% RSLogix 500 project IIS REV 1.0. 4.29.16.RSS, saved by version 10.00.00.00 %
PROJECT "IISM1200"    % processor: MicroLogix 1200 %

PROGRAM FILES
  LAD 2 "MAIN_PROG"  27 rungs

DATA FILES
  O0 OUTPUT  4 elements
  I1 INPUT  4 elements
  S2 STATUS  66 elements
  B3 BINARY  2 elements
  T4 TIMER  4 elements
  C5 COUNTER  1 elements
  R6 CONTROL  1 elements
  N7 INTEGER  1 elements
  F8 FLOAT  1 elements

LADDER 2 "MAIN_PROG"
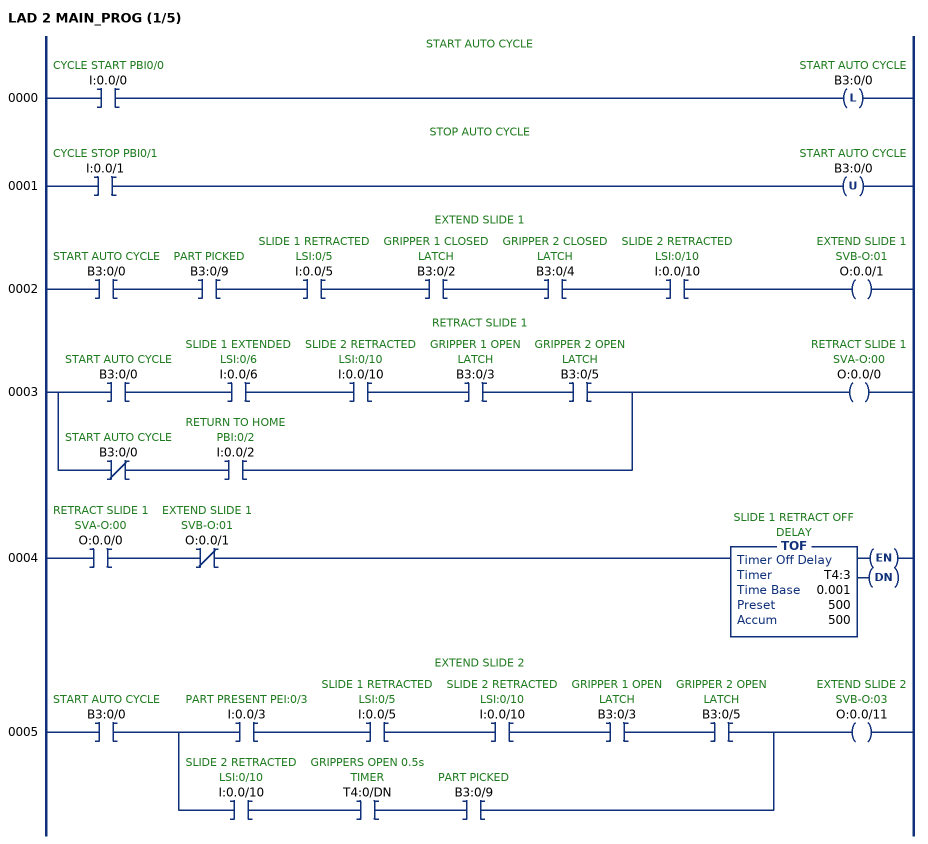
% Rung: 0 %
% START AUTO CYCLE %
SOR XIC I:0.0/0 OTL B3:0/0 EOR
%   I:0.0/0  "CYCLE START PBI0/0" %
%   B3:0/0  "START AUTO CYCLE" %
% Rung: 1 %
% STOP AUTO CYCLE %
SOR XIC I:0.0/1 OTU B3:0/0 EOR
%   I:0.0/1  "CYCLE STOP PBI0/1" %
%   B3:0/0  "START AUTO CYCLE" %
% Rung: 2 %
% EXTEND SLIDE 1 %
SOR XIC B3:0/0 XIC B3:0/9 XIC I:0.0/5 XIC B3:0/2 XIC B3:0/4 XIC I:0.0/10 OTE O:0.0/1 EOR
%   B3:0/0  "START AUTO CYCLE" %
%   B3:0/9  "PART PICKED" %
%   I:0.0/5  "SLIDE 1 RETRACTED LSI:0/5" %
%   B3:0/2  "GRIPPER 1 CLOSED LATCH" %
%   B3:0/4  "GRIPPER 2 CLOSED LATCH" %
%   I:0.0/10  "SLIDE 2 RETRACTED LSI:0/10" %
%   O:0.0/1  "EXTEND SLIDE 1 SVB-O:01" %
% Rung: 3 %
% RETRACT SLIDE 1 %
SOR BST XIC B3:0/0 XIC I:0.0/6 XIC I:0.0/10 XIC B3:0/3 XIC B3:0/5 NXB XIO B3:0/0 XIC I:0.0/2 BND OTE O:0.0/0 EOR
%   B3:0/0  "START AUTO CYCLE" %
%   I:0.0/6  "SLIDE 1 EXTENDED LSI:0/6" %
%   I:0.0/10  "SLIDE 2 RETRACTED LSI:0/10" %
%   B3:0/3  "GRIPPER 1 OPEN LATCH" %
%   B3:0/5  "GRIPPER 2 OPEN LATCH" %
%   I:0.0/2  "RETURN TO HOME PBI:0/2" %
%   O:0.0/0  "RETRACT SLIDE 1 SVA-O:00" %
% Rung: 4 %
SOR XIC O:0.0/0 XIO O:0.0/1 TOF T4:3 0.001 500 500 EOR
%   O:0.0/0  "RETRACT SLIDE 1 SVA-O:00" %
%   O:0.0/1  "EXTEND SLIDE 1 SVB-O:01" %
%   T4:3  "SLIDE 1 RETRACT OFF DELAY" %
% Rung: 5 %
% EXTEND SLIDE 2 %
SOR XIC B3:0/0 BST XIC I:0.0/3 XIC I:0.0/5 XIC I:0.0/10 XIC B3:0/3 XIC B3:0/5 NXB XIC I:0.0/10 XIC T4:0/DN XIC B3:0/9 BND OTE O:0.0/11 EOR
%   B3:0/0  "START AUTO CYCLE" %
%   I:0.0/3  "PART PRESENT PEI:0/3" %
%   I:0.0/5  "SLIDE 1 RETRACTED LSI:0/5" %
%   I:0.0/10  "SLIDE 2 RETRACTED LSI:0/10" %
%   B3:0/3  "GRIPPER 1 OPEN LATCH" %
%   B3:0/5  "GRIPPER 2 OPEN LATCH" %
%   T4:0  "GRIPPERS OPEN 0.5s TIMER" %
%   B3:0/9  "PART PICKED" %
%   O:0.0/11  "EXTEND SLIDE 2 SVB-O:03" %

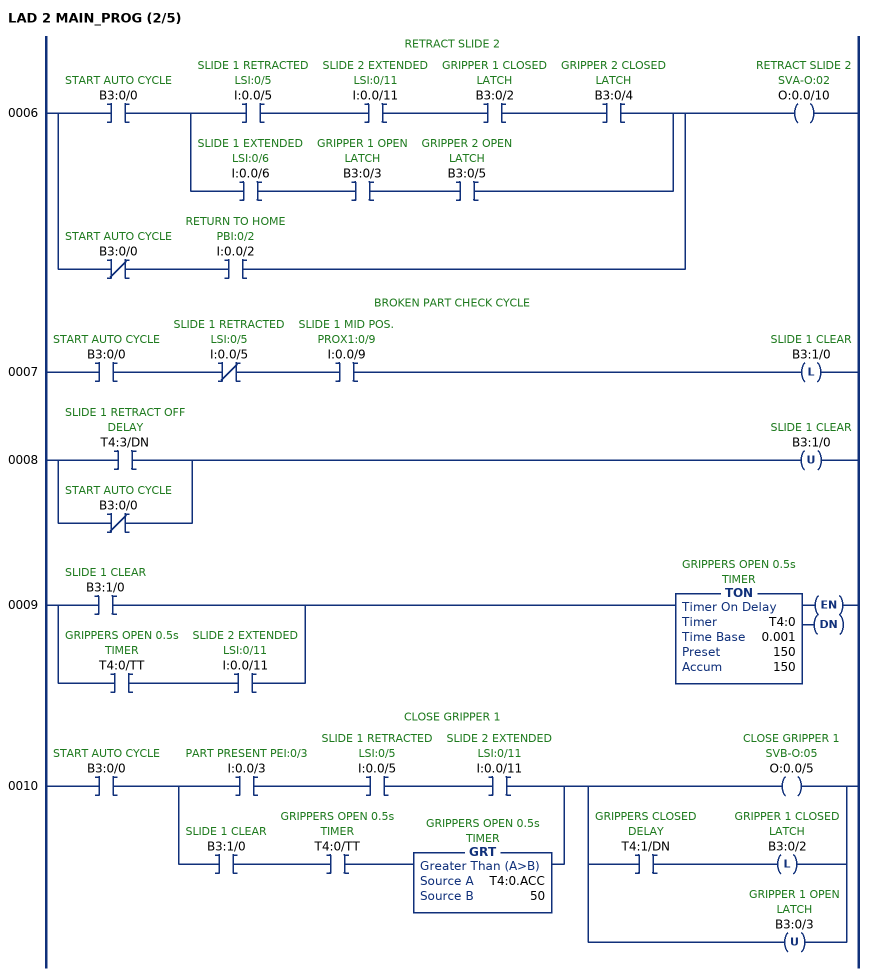
% Rung: 6 %
% RETRACT SLIDE 2 %
SOR BST XIC B3:0/0 BST XIC I:0.0/5 XIC I:0.0/11 XIC B3:0/2 XIC B3:0/4 NXB XIC I:0.0/6 XIC B3:0/3 XIC B3:0/5 BND NXB XIO B3:0/0 XIC I:0.0/2 BND OTE O:0.0/10 EOR
%   B3:0/0  "START AUTO CYCLE" %
%   I:0.0/5  "SLIDE 1 RETRACTED LSI:0/5" %
%   I:0.0/11  "SLIDE 2 EXTENDED LSI:0/11" %
%   B3:0/2  "GRIPPER 1 CLOSED LATCH" %
%   B3:0/4  "GRIPPER 2 CLOSED LATCH" %
%   I:0.0/6  "SLIDE 1 EXTENDED LSI:0/6" %
%   B3:0/3  "GRIPPER 1 OPEN LATCH" %
%   B3:0/5  "GRIPPER 2 OPEN LATCH" %
%   I:0.0/2  "RETURN TO HOME PBI:0/2" %
%   O:0.0/10  "RETRACT SLIDE 2 SVA-O:02" %
% Rung: 7 %
% BROKEN PART CHECK CYCLE %
SOR XIC B3:0/0 XIO I:0.0/5 XIC I:0.0/9 OTL B3:1/0 EOR
%   B3:0/0  "START AUTO CYCLE" %
%   I:0.0/5  "SLIDE 1 RETRACTED LSI:0/5" %
%   I:0.0/9  "SLIDE 1 MID POS. PROX1:0/9" %
%   B3:1/0  "SLIDE 1 CLEAR" %
% Rung: 8 %
SOR BST XIC T4:3/DN NXB XIO B3:0/0 BND OTU B3:1/0 EOR
%   T4:3  "SLIDE 1 RETRACT OFF DELAY" %
%   B3:0/0  "START AUTO CYCLE" %
%   B3:1/0  "SLIDE 1 CLEAR" %
% Rung: 9 %
SOR BST XIC B3:1/0 NXB XIC T4:0/TT XIC I:0.0/11 BND TON T4:0 0.001 150 150 EOR
%   B3:1/0  "SLIDE 1 CLEAR" %
%   T4:0  "GRIPPERS OPEN 0.5s TIMER" %
%   I:0.0/11  "SLIDE 2 EXTENDED LSI:0/11" %
% Rung: 10 %
% CLOSE GRIPPER 1 %
SOR XIC B3:0/0 BST XIC I:0.0/3 XIC I:0.0/5 XIC I:0.0/11 NXB XIC B3:1/0 XIC T4:0/TT GRT T4:0.ACC 50 BND BST OTE O:0.0/5 NXB XIC T4:1/DN OTL B3:0/2 NXB OTU B3:0/3 BND EOR
%   B3:0/0  "START AUTO CYCLE" %
%   I:0.0/3  "PART PRESENT PEI:0/3" %
%   I:0.0/5  "SLIDE 1 RETRACTED LSI:0/5" %
%   I:0.0/11  "SLIDE 2 EXTENDED LSI:0/11" %
%   B3:1/0  "SLIDE 1 CLEAR" %
%   T4:0  "GRIPPERS OPEN 0.5s TIMER" %
%   O:0.0/5  "CLOSE GRIPPER 1 SVB-O:05" %
%   T4:1/DN  "GRIPPERS CLOSED DELAY" %
%   B3:0/2  "GRIPPER 1 CLOSED LATCH" %
%   B3:0/3  "GRIPPER 1 OPEN LATCH" %

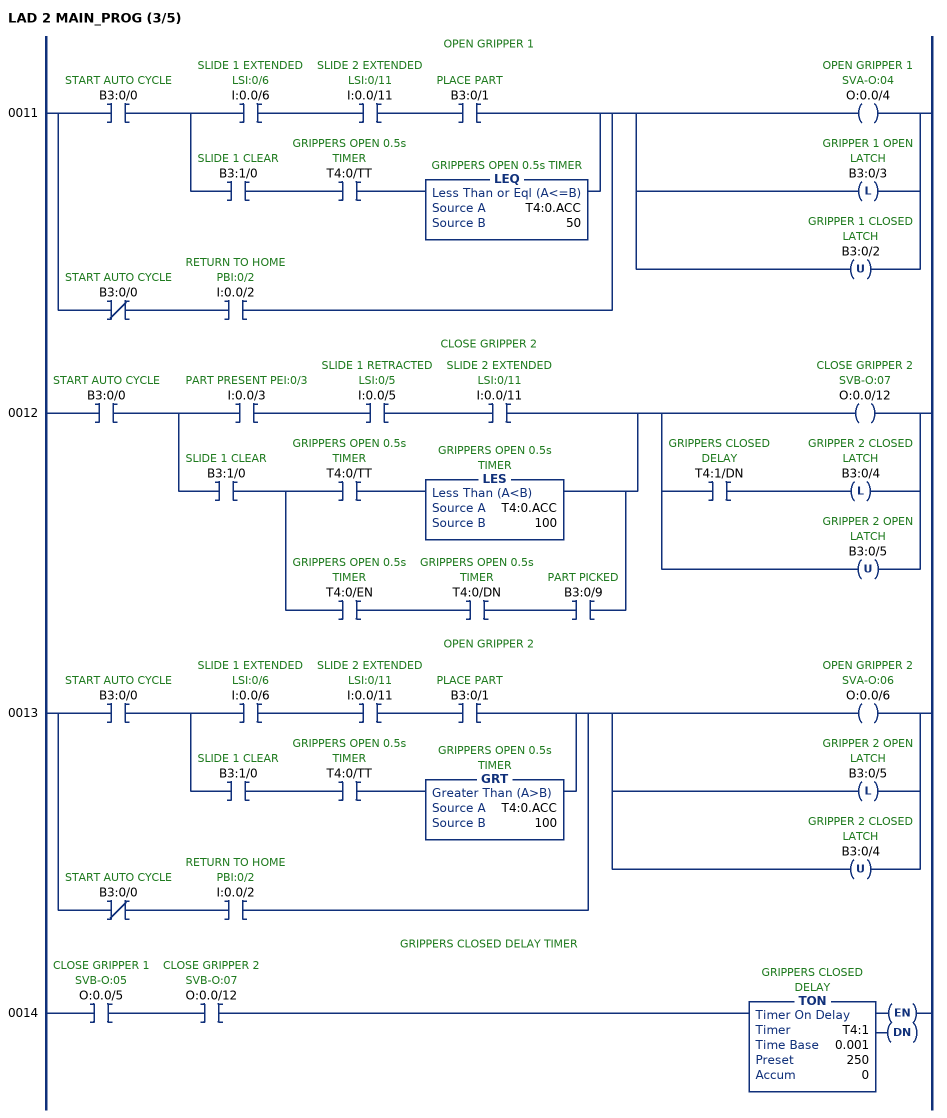
% Rung: 11 %
% OPEN GRIPPER 1 %
SOR BST XIC B3:0/0 BST XIC I:0.0/6 XIC I:0.0/11 XIC B3:0/1 NXB XIC B3:1/0 XIC T4:0/TT LEQ T4:0.ACC 50 BND NXB XIO B3:0/0 XIC I:0.0/2 BND BST OTE O:0.0/4 NXB OTL B3:0/3 NXB OTU B3:0/2 BND EOR
%   B3:0/0  "START AUTO CYCLE" %
%   I:0.0/6  "SLIDE 1 EXTENDED LSI:0/6" %
%   I:0.0/11  "SLIDE 2 EXTENDED LSI:0/11" %
%   B3:0/1  "PLACE PART" %
%   B3:1/0  "SLIDE 1 CLEAR" %
%   T4:0  "GRIPPERS OPEN 0.5s TIMER" %
%   I:0.0/2  "RETURN TO HOME PBI:0/2" %
%   O:0.0/4  "OPEN GRIPPER 1 SVA-O:04" %
%   B3:0/3  "GRIPPER 1 OPEN LATCH" %
%   B3:0/2  "GRIPPER 1 CLOSED LATCH" %
% Rung: 12 %
% CLOSE GRIPPER 2 %
SOR XIC B3:0/0 BST XIC I:0.0/3 XIC I:0.0/5 XIC I:0.0/11 NXB XIC B3:1/0 BST XIC T4:0/TT LES T4:0.ACC 100 NXB XIC T4:0/EN XIC T4:0/DN XIC B3:0/9 BND BND BST OTE O:0.0/12 NXB XIC T4:1/DN OTL B3:0/4 NXB OTU B3:0/5 BND EOR
%   B3:0/0  "START AUTO CYCLE" %
%   I:0.0/3  "PART PRESENT PEI:0/3" %
%   I:0.0/5  "SLIDE 1 RETRACTED LSI:0/5" %
%   I:0.0/11  "SLIDE 2 EXTENDED LSI:0/11" %
%   B3:1/0  "SLIDE 1 CLEAR" %
%   T4:0  "GRIPPERS OPEN 0.5s TIMER" %
%   B3:0/9  "PART PICKED" %
%   O:0.0/12  "CLOSE GRIPPER 2 SVB-O:07" %
%   T4:1/DN  "GRIPPERS CLOSED DELAY" %
%   B3:0/4  "GRIPPER 2 CLOSED LATCH" %
%   B3:0/5  "GRIPPER 2 OPEN LATCH" %
% Rung: 13 %
% OPEN GRIPPER 2 %
SOR BST XIC B3:0/0 BST XIC I:0.0/6 XIC I:0.0/11 XIC B3:0/1 NXB XIC B3:1/0 XIC T4:0/TT GRT T4:0.ACC 100 BND NXB XIO B3:0/0 XIC I:0.0/2 BND BST OTE O:0.0/6 NXB OTL B3:0/5 NXB OTU B3:0/4 BND EOR
%   B3:0/0  "START AUTO CYCLE" %
%   I:0.0/6  "SLIDE 1 EXTENDED LSI:0/6" %
%   I:0.0/11  "SLIDE 2 EXTENDED LSI:0/11" %
%   B3:0/1  "PLACE PART" %
%   B3:1/0  "SLIDE 1 CLEAR" %
%   T4:0  "GRIPPERS OPEN 0.5s TIMER" %
%   I:0.0/2  "RETURN TO HOME PBI:0/2" %
%   O:0.0/6  "OPEN GRIPPER 2 SVA-O:06" %
%   B3:0/5  "GRIPPER 2 OPEN LATCH" %
%   B3:0/4  "GRIPPER 2 CLOSED LATCH" %
% Rung: 14 %
% GRIPPERS CLOSED DELAY TIMER %
SOR XIC O:0.0/5 XIC O:0.0/12 TON T4:1 0.001 250 0 EOR
%   O:0.0/5  "CLOSE GRIPPER 1 SVB-O:05" %
%   O:0.0/12  "CLOSE GRIPPER 2 SVB-O:07" %
%   T4:1  "GRIPPERS CLOSED DELAY" %

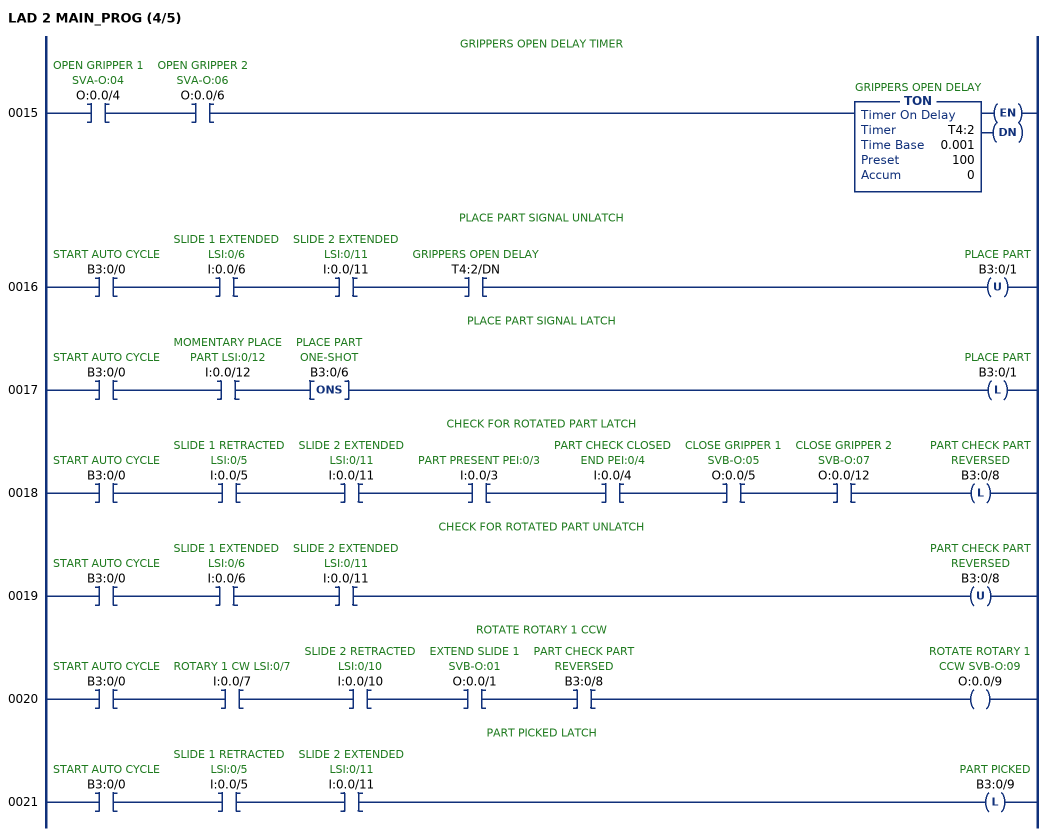
% Rung: 15 %
% GRIPPERS OPEN DELAY TIMER %
SOR XIC O:0.0/4 XIC O:0.0/6 TON T4:2 0.001 100 0 EOR
%   O:0.0/4  "OPEN GRIPPER 1 SVA-O:04" %
%   O:0.0/6  "OPEN GRIPPER 2 SVA-O:06" %
%   T4:2  "GRIPPERS OPEN DELAY" %
% Rung: 16 %
% PLACE PART SIGNAL UNLATCH %
SOR XIC B3:0/0 XIC I:0.0/6 XIC I:0.0/11 XIC T4:2/DN OTU B3:0/1 EOR
%   B3:0/0  "START AUTO CYCLE" %
%   I:0.0/6  "SLIDE 1 EXTENDED LSI:0/6" %
%   I:0.0/11  "SLIDE 2 EXTENDED LSI:0/11" %
%   T4:2  "GRIPPERS OPEN DELAY" %
%   B3:0/1  "PLACE PART" %
% Rung: 17 %
% PLACE PART SIGNAL LATCH %
SOR XIC B3:0/0 XIC I:0.0/12 ONS B3:0/6 OTL B3:0/1 EOR
%   B3:0/0  "START AUTO CYCLE" %
%   I:0.0/12  "MOMENTARY PLACE PART LSI:0/12" %
%   B3:0/6  "PLACE PART ONE-SHOT" %
%   B3:0/1  "PLACE PART" %
% Rung: 18 %
% CHECK FOR ROTATED PART LATCH %
SOR XIC B3:0/0 XIC I:0.0/5 XIC I:0.0/11 XIC I:0.0/3 XIC I:0.0/4 XIC O:0.0/5 XIC O:0.0/12 OTL B3:0/8 EOR
%   B3:0/0  "START AUTO CYCLE" %
%   I:0.0/5  "SLIDE 1 RETRACTED LSI:0/5" %
%   I:0.0/11  "SLIDE 2 EXTENDED LSI:0/11" %
%   I:0.0/3  "PART PRESENT PEI:0/3" %
%   I:0.0/4  "PART CHECK CLOSED END PEI:0/4" %
%   O:0.0/5  "CLOSE GRIPPER 1 SVB-O:05" %
%   O:0.0/12  "CLOSE GRIPPER 2 SVB-O:07" %
%   B3:0/8  "PART CHECK PART REVERSED" %
% Rung: 19 %
% CHECK FOR ROTATED PART UNLATCH %
SOR XIC B3:0/0 XIC I:0.0/6 XIC I:0.0/11 OTU B3:0/8 EOR
%   B3:0/0  "START AUTO CYCLE" %
%   I:0.0/6  "SLIDE 1 EXTENDED LSI:0/6" %
%   I:0.0/11  "SLIDE 2 EXTENDED LSI:0/11" %
%   B3:0/8  "PART CHECK PART REVERSED" %
% Rung: 20 %
% ROTATE ROTARY 1 CCW %
SOR XIC B3:0/0 XIC I:0.0/7 XIC I:0.0/10 XIC O:0.0/1 XIC B3:0/8 OTE O:0.0/9 EOR
%   B3:0/0  "START AUTO CYCLE" %
%   I:0.0/7  "ROTARY 1 CW LSI:0/7" %
%   I:0.0/10  "SLIDE 2 RETRACTED LSI:0/10" %
%   O:0.0/1  "EXTEND SLIDE 1 SVB-O:01" %
%   B3:0/8  "PART CHECK PART REVERSED" %
%   O:0.0/9  "ROTATE ROTARY 1 CCW SVB-O:09" %
% Rung: 21 %
% PART PICKED LATCH %
SOR XIC B3:0/0 XIC I:0.0/5 XIC I:0.0/11 OTL B3:0/9 EOR
%   B3:0/0  "START AUTO CYCLE" %
%   I:0.0/5  "SLIDE 1 RETRACTED LSI:0/5" %
%   I:0.0/11  "SLIDE 2 EXTENDED LSI:0/11" %
%   B3:0/9  "PART PICKED" %

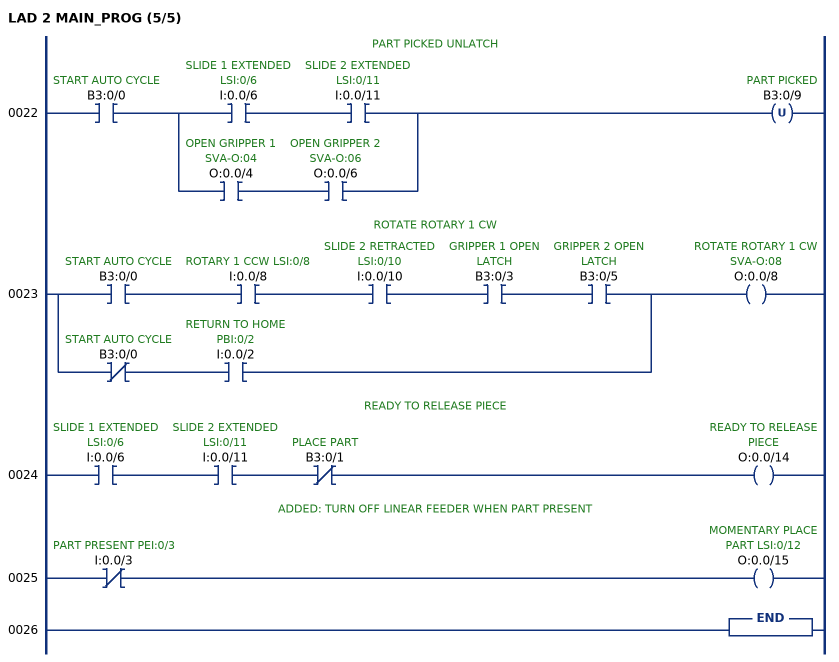
% Rung: 22 %
% PART PICKED UNLATCH %
SOR XIC B3:0/0 BST XIC I:0.0/6 XIC I:0.0/11 NXB XIC O:0.0/4 XIC O:0.0/6 BND OTU B3:0/9 EOR
%   B3:0/0  "START AUTO CYCLE" %
%   I:0.0/6  "SLIDE 1 EXTENDED LSI:0/6" %
%   I:0.0/11  "SLIDE 2 EXTENDED LSI:0/11" %
%   O:0.0/4  "OPEN GRIPPER 1 SVA-O:04" %
%   O:0.0/6  "OPEN GRIPPER 2 SVA-O:06" %
%   B3:0/9  "PART PICKED" %
% Rung: 23 %
% ROTATE ROTARY 1 CW %
SOR BST XIC B3:0/0 XIC I:0.0/8 XIC I:0.0/10 XIC B3:0/3 XIC B3:0/5 NXB XIO B3:0/0 XIC I:0.0/2 BND OTE O:0.0/8 EOR
%   B3:0/0  "START AUTO CYCLE" %
%   I:0.0/8  "ROTARY 1 CCW LSI:0/8" %
%   I:0.0/10  "SLIDE 2 RETRACTED LSI:0/10" %
%   B3:0/3  "GRIPPER 1 OPEN LATCH" %
%   B3:0/5  "GRIPPER 2 OPEN LATCH" %
%   I:0.0/2  "RETURN TO HOME PBI:0/2" %
%   O:0.0/8  "ROTATE ROTARY 1 CW SVA-O:08" %
% Rung: 24 %
% READY TO RELEASE PIECE %
SOR XIC I:0.0/6 XIC I:0.0/11 XIO B3:0/1 OTE O:0.0/14 EOR
%   I:0.0/6  "SLIDE 1 EXTENDED LSI:0/6" %
%   I:0.0/11  "SLIDE 2 EXTENDED LSI:0/11" %
%   B3:0/1  "PLACE PART" %
%   O:0.0/14  "READY TO RELEASE PIECE" %
% Rung: 25 %
% ADDED: TURN OFF LINEAR FEEDER WHEN PART PRESENT %
SOR XIO I:0.0/3 OTE O:0.0/15 EOR
%   I:0.0/3  "PART PRESENT PEI:0/3" %
%   O:0.0/15  "MOMENTARY PLACE PART LSI:0/12" %
% Rung: 26 %
SOR END EOR

OTHER DOCUMENTED ADDRESSES
  DFILE:0  "OUTPUT"
  DFILE:1  "INPUT"
  DFILE:2  "STATUS"
  DFILE:3  "BINARY"
  DFILE:4  "TIMER"
  DFILE:5  "COUNTER"
  DFILE:6  "CONTROL"
  DFILE:7  "INTEGER"
  DFILE:8  "FLOAT"
  I:0  "CYCLE START PBI0/0"

COMMENTS NOT ATTACHED TO A CURRENT RUNG
  B3:0/0: START AUTO CYCLE

DATA TABLE (non-zero values as saved)
DATA B3
% B3:0 % 0X0001 0X0001
DATA T4
% .PRE .ACC %
% T4:0 % 150 150
% T4:1 % 250 0
% T4:2 % 100 0
% T4:3 % 500 500
